// TIA Portal V18 export
TYPE "UDT_FrostProtection"
// stored: IsFailsafeCompliant false
   STRUCT
      AlarmWaterTempLimit : Array[1..3] of Real;
      BandMin : Array[1..3] of Real;
      BandMax : Array[1..3] of Real;
      OATMin : Array[1..3] of Real;
      OATMax : Array[1..3] of Real;
      CalculatedAddition : Array[1..3] of Real;
      OATtoStartPreheating : Array[1..3] of Real;
   END_STRUCT;
END_TYPE
